// SIMATIC STEP 7 (V5.x) project waterplant
// CPU: CPU 314C-2 DP
// station: Hardware
// station: SIMATIC 300(1)
// station: P_ADR_BUS
// station: P_ADR_BUS
// station: Configuration
// program: S7 Program(1)

SYMBOL_TABLE
"S5TI_TIM"	FC 33	FC 33	// S5 Time to IEC Time
"TIM_S5TI"	FC 40	FC 40	// IEC Time to S5 Time
"SCALE"	FC 105	FC 105	// Scaling Values
"start system"	I 0.0	BOOL
"LEVsensor Raw tank"	I 0.1	BOOL
"raw pump run feedback"	I 0.2	BOOL
"low filter tank1"	I 0.3	BOOL
"high filter tank1"	I 0.4	BOOL
"low filter tank2"	I 0.5	BOOL
"emergency pressed"	I 0.6	BOOL
"sludge H-sensor tank"	I 0.7	BOOL
"LEVsensor flash mixer"	I 1.0	BOOL
"LEVsensor slow mixer"	I 1.1	BOOL
"LEVsenclarifier buttom"	I 1.2	BOOL
"sludge L-sensor tank"	I 1.3	BOOL
"led photo sensor"	I 1.4	BOOL
"service intake"	I 1.5	BOOL
"flash mixer feedback"	I 2.0	BOOL
"slow mixer feedback"	I 2.1	BOOL
"clarifier feedback"	I 2.2	BOOL
"blower feedback"	I 2.3	BOOL
"wash water feedback"	I 2.4	BOOL
"flash mixer over sensor"	I 2.5	BOOL
"PLC OK"	M 0.0	BOOL
"reset sludge clarifier"	M 0.1	BOOL
"sludge clarifier relay"	M 0.2	BOOL
"test clarifier from scad"	M 0.3	BOOL
"test raw pump scada"	M 0.4	BOOL
"test flash mixer scada"	M 0.5	BOOL
"test slow mixer scada"	M 0.6	BOOL
"test sludge pump scada"	M 0.7	BOOL
"sludge pipe color scada"	M 1.0	BOOL
"led test from scada"	M 1.1	BOOL
"air valve relay"	M 1.2	BOOL
"air valve test scada"	M 1.3	BOOL
"traet pipe color"	M 1.4	BOOL
"wash water relay"	M 1.5	BOOL
"wash water test scada"	M 1.6	BOOL
"zero washing time messag"	M 1.7	BOOL
"sludge time message"	M 2.0	BOOL
"reset alarm scada"	M 2.1	BOOL
"reset hardware alarm"	M 2.2	BOOL
"alarm on scada"	M 2.3	BOOL
"factory reset scada"	M 2.4	BOOL
"system run for scada"	M 2.5	BOOL
"filter tank H-L relay"	M 2.6	BOOL
"sludge pump relay"	M 2.7	BOOL
"raw pump feedback alarm"	M 3.0	BOOL
"force stop raw pump"	M 3.1	BOOL
"force stop AL2SO4"	M 3.2	BOOL
"force stop flash mixer"	M 3.3	BOOL
"force stop slow mixer"	M 3.4	BOOL
"force stop sludge pump"	M 3.5	BOOL
"force stop clarifier"	M 3.6	BOOL
"air blower force stop"	M 3.7	BOOL
"wash pump force stop"	M 4.0	BOOL
"alarm on scada relay"	M 4.1	BOOL
"air valve relay 2"	M 4.2	BOOL
"wash water relay 2"	M 4.3	BOOL
"force stop light"	M 4.4	BOOL
"flash mixer over"	M 4.6	BOOL
"zero analog bibolar"	M 5.0	BOOL
"flash mixer tank full"	M 5.1	BOOL
"slow mixer full tank"	M 5.2	BOOL
"flash feedback  alarm"	M 5.3	BOOL
"start reverse now scada"	M 5.5	BOOL
"restart reverse wash sca"	M 5.6	BOOL
"No restert scada"	M 5.7	BOOL
"No restart marker"	M 6.0	BOOL
"reverse wash wait messag"	M 6.1	BOOL
"sludge tank filling"	M 6.2	BOOL
"emeergency mode for scad"	M 6.3	BOOL
"start now marker"	M 6.4	BOOL
"reverse wash has started"	M 6.6	BOOL
"slow feedback alarm"	M 6.7	BOOL
"clarifier feedback alarm"	M 7.0	BOOL
"blower feedback alarm"	M 7.1	BOOL
"wash feedback alarm"	M 7.2	BOOL
"flash over flow alarm"	M 7.3	BOOL
"y.restart rev wash scada"	M 8.0	BOOL
"reverser timer reminder"	MD 210	DWORD
"rev wash reminder scada"	MD 212	DWORD
"sludge clarifier off sca"	MW 50	WORD
"sludge clarifier on sca"	MW 80	WORD
"reverse wash time scada"	MW 150	WORD
"voltage sensor analoge"	PIW 3	WORD
"current sensor analoge"	PIW 5	WORD
"raw pump"	Q 0.0	BOOL
"AL2SO4 valve"	Q 0.1	BOOL
"flash mixer"	Q 0.2	BOOL
"slow mixer"	Q 0.3	BOOL
"sludge motor clarifier"	Q 0.4	BOOL
"enter valve filter1"	Q 0.5	BOOL
"enter valve filter2"	Q 0.6	BOOL
"treat1"	Q 0.7	BOOL
"treat2"	Q 1.0	BOOL
"air valve1"	Q 1.1	BOOL
"wash water1"	Q 1.2	BOOL
"sludge pump"	Q 1.3	BOOL
"alarm"	Q 1.4	BOOL
"led"	Q 1.5	BOOL
"sludge valve filter1"	Q 1.6	BOOL
"sludge valve filter2"	Q 1.7	BOOL
"TON"	SFB 4	SFB 4	// Generate an On Delay
"AL2SO4 open time"	T 1	TIMER
"clarifier off time"	T 2	TIMER
"clarifier on time"	T 3	TIMER
"high treat tank dist"	T 4	TIMER
"wash timer process"	T 5	TIMER
"air valve timer"	T 6	TIMER
"before wash time"	T 8	TIMER	// delay time before start washing
"treat1 dist"	T 9	TIMER
"enter valve 1 delay time"	T 10	TIMER
"slow feedback timer"	T 11	TIMER
"delay time before alarm"	T 12	TIMER
"factory reset timer"	T 13	TIMER
"start system timer"	T 14	TIMER
"clarifier feedback timer"	T 15	TIMER
"blower feedback timer"	T 16	TIMER
"sludge pump force stop t"	T 17	TIMER
"clarifier force stop t"	T 18	TIMER
"raw pump force stop t"	T 19	TIMER
"clarifier before start t"	T 20	TIMER
"timer before wash proces"	T 21	TIMER
"wash feedback timer"	T 22	TIMER
"treat 2 dist."	T 23	TIMER
"flash mixer feedback tim"	T 24	TIMER
"raw pump feedback timer"	T 25	TIMER
"enter valve 2 timer"	T 26	TIMER
"before restart message"	T 30	TIMER
"rewash wait alarm timer"	T 31	TIMER
END_SYMBOL_TABLE

// FC 33: know-how protected block, not included

// FC 40: know-how protected block, not included

// FC 105: know-how protected block, not included

ORGANIZATION_BLOCK OB 1
TITLE = "Main Program Sweep (Cycle)"
VERSION : 0.1
VAR_TEMP
  OB1_EV_CLASS : BYTE ;	//Bits 0-3 = 1 (Coming event), Bits 4-7 = 1 (Event class 1)
  OB1_SCAN_1 : BYTE ;	//1 (Cold restart scan 1 of OB 1), 3 (Scan 2-n of OB 1)
  OB1_PRIORITY : BYTE ;	//Priority of OB Execution
  OB1_OB_NUMBR : BYTE ;	//1 (Organization block 1, OB1)
  OB1_RESERVED_1 : BYTE ;	//Reserved for system
  OB1_RESERVED_2 : BYTE ;	//Reserved for system
  OB1_PREV_CYCLE : INT ;	//Cycle time of previous OB1 scan (milliseconds)
  OB1_MIN_CYCLE : INT ;	//Minimum cycle time of OB1 (milliseconds)
  OB1_MAX_CYCLE : INT ;	//Maximum cycle time of OB1 (milliseconds)
  OB1_DATE_TIME : DATE_AND_TIME ;	//Date and time OB1 started
END_VAR
BEGIN
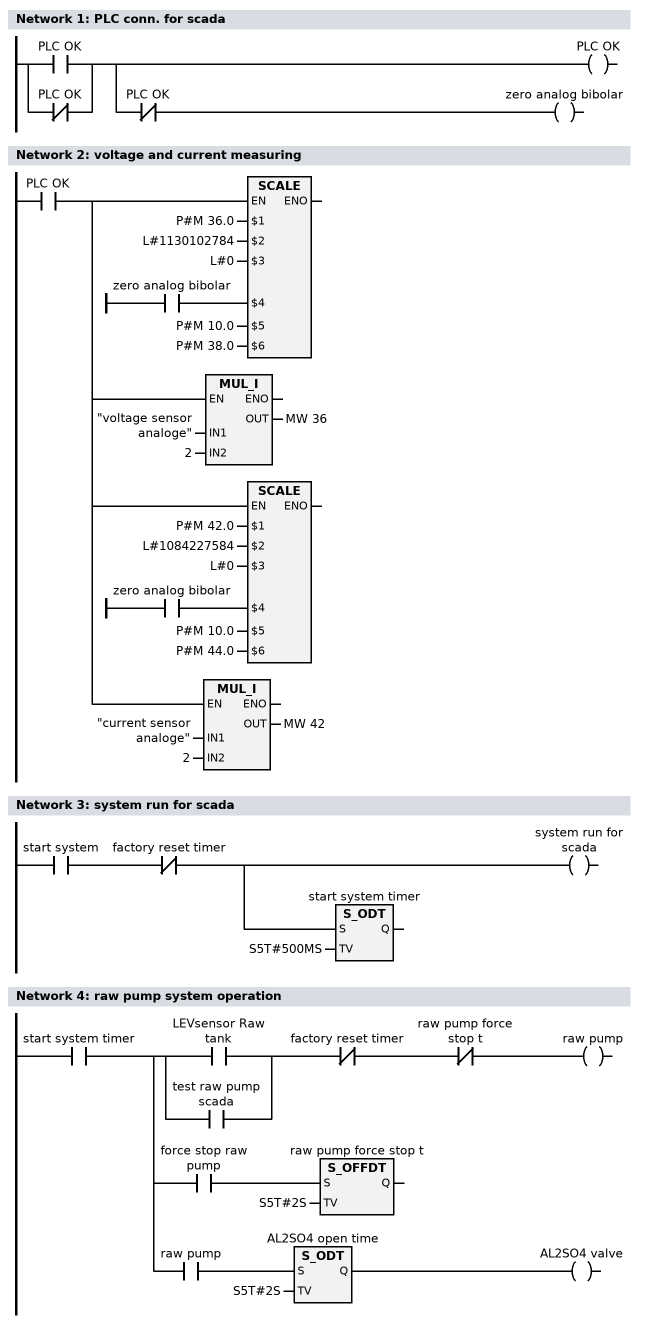
NETWORK
TITLE = PLC conn. for scada
      O     "PLC OK";
      ON    "PLC OK";
      =     L 240.0;
      A     L 240.0;
      BLD   102;
      =     "PLC OK";
      A     L 240.0;
      AN    "PLC OK";
      =     "zero analog bibolar";
NETWORK
TITLE = voltage and current measuring
      A     "PLC OK";
      =     L 240.0;
      A     "zero analog bibolar";
      =     L 240.1;
      BLD   103;
      A     L 240.0;
      JNB   _001;
      CALL  "SCALE" (
           $1                       := P#M 36.0,
           $2                       := L#1130102784,
           $3                       := L#0,
           $4                       := L 240.1,
           $5                       := P#M 10.0,
           $6                       := P#M 38.0);
_001: NOP   0;
      A     L 240.0;
      JNB   _002;
      L     "voltage sensor analoge";
      L     2;
      *I;
      T     MW 36;
_002: NOP   0;
      A     "zero analog bibolar";
      =     L 240.1;
      BLD   103;
      A     L 240.0;
      JNB   _003;
      CALL  "SCALE" (
           $1                       := P#M 42.0,
           $2                       := L#1084227584,
           $3                       := L#0,
           $4                       := L 240.1,
           $5                       := P#M 10.0,
           $6                       := P#M 44.0);
_003: NOP   0;
      A     L 240.0;
      JNB   _004;
      L     "current sensor analoge";
      L     2;
      *I;
      T     MW 42;
_004: NOP   0;
NETWORK
TITLE = system run for scada
      A     "start system";
      AN    "factory reset timer";
      =     L 240.0;
      A     L 240.0;
      BLD   102;
      =     "system run for scada";
      A     L 240.0;
      L     S5T#500MS;
      SD    "start system timer";
      NOP   0;
      NOP   0;
      NOP   0;
      NOP   0;
NETWORK
TITLE = raw pump system operation
      A     "start system timer";
      =     L 240.0;
      A     L 240.0;
      A(;
      O     "LEVsensor Raw tank";
      O     "test raw pump scada";
      );
      AN    "factory reset timer";
      AN    "raw pump force stop t";
      =     "raw pump";
      A     L 240.0;
      A     "force stop raw pump";
      L     S5T#2S;
      SF    "raw pump force stop t";
      NOP   0;
      NOP   0;
      NOP   0;
      NOP   0;
      A     L 240.0;
      A     "raw pump";
      L     S5T#2S;
      SD    "AL2SO4 open time";
      NOP   0;
      NOP   0;
      NOP   0;
      A     "AL2SO4 open time";
      =     "AL2SO4 valve";
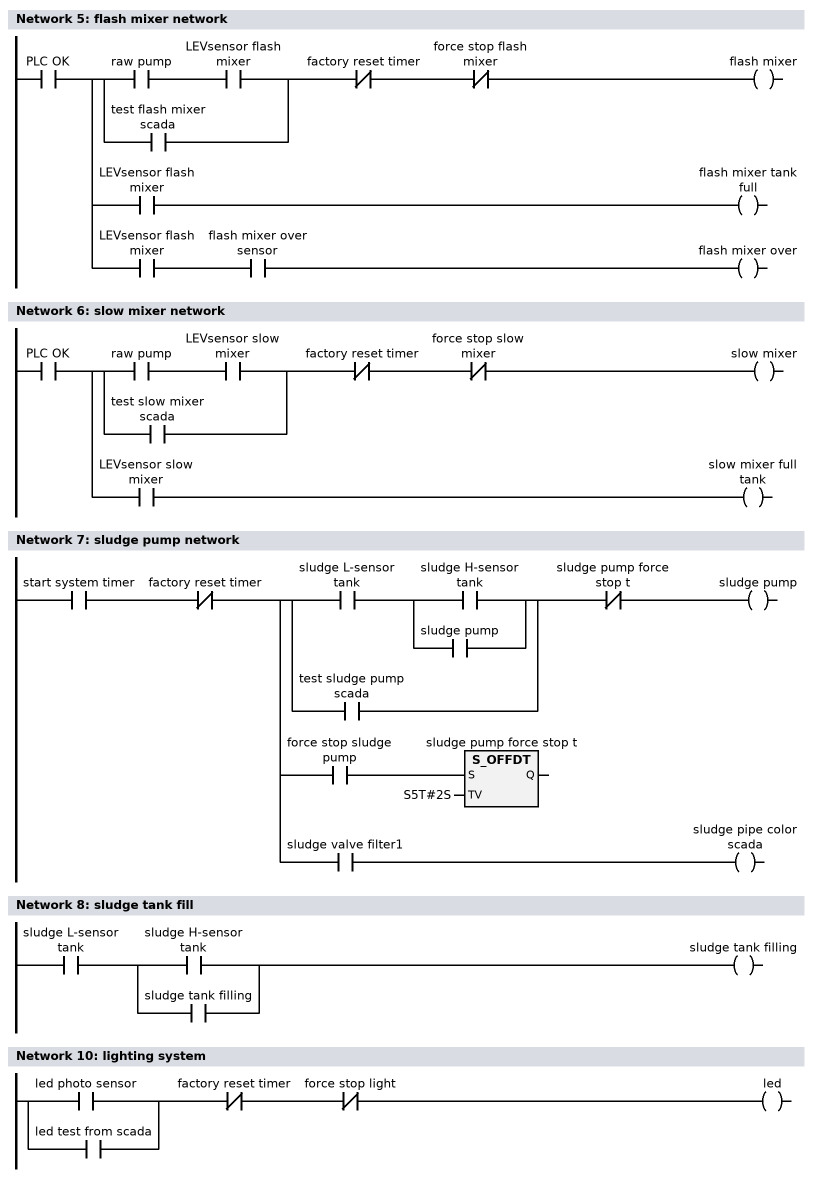
NETWORK
TITLE = flash mixer network
      A     "PLC OK";
      =     L 240.0;
      A     L 240.0;
      A(;
      A     "raw pump";
      A     "LEVsensor flash mixer";
      O     "test flash mixer scada";
      );
      AN    "factory reset timer";
      AN    "force stop flash mixer";
      =     "flash mixer";
      A     L 240.0;
      A     "LEVsensor flash mixer";
      =     "flash mixer tank full";
      A     L 240.0;
      A     "LEVsensor flash mixer";
      A     "flash mixer over sensor";
      =     "flash mixer over";
NETWORK
TITLE = slow mixer network
      A     "PLC OK";
      =     L 240.0;
      A     L 240.0;
      A(;
      A     "raw pump";
      A     "LEVsensor slow mixer";
      O     "test slow mixer scada";
      );
      AN    "factory reset timer";
      AN    "force stop slow mixer";
      =     "slow mixer";
      A     L 240.0;
      A     "LEVsensor slow mixer";
      =     "slow mixer full tank";
NETWORK
TITLE = sludge pump network
      A     "start system timer";
      AN    "factory reset timer";
      =     L 240.0;
      A     L 240.0;
      A(;
      A     "sludge L-sensor tank";
      A(;
      O     "sludge H-sensor tank";
      O     "sludge pump";
      );
      O     "test sludge pump scada";
      );
      AN    "sludge pump force stop t";
      =     "sludge pump";
      A     L 240.0;
      A     "force stop sludge pump";
      L     S5T#2S;
      SF    "sludge pump force stop t";
      NOP   0;
      NOP   0;
      NOP   0;
      NOP   0;
      A     L 240.0;
      A     "sludge valve filter1";
      =     "sludge pipe color scada";
NETWORK
TITLE = sludge tank fill
      A     "sludge L-sensor tank";
      A(;
      O     "sludge H-sensor tank";
      O     "sludge tank filling";
      );
      =     "sludge tank filling";
NETWORK
TITLE = sludge motor clarifier timer operation
      A     "start system timer";
      =     L 240.0;
      A     L 240.0;
      A     "raw pump";
      A     "LEVsenclarifier buttom";
      AN    "factory reset timer";
      =     L 240.1;
      A(;
      A     L 240.1;
      A(;
      L     "sludge clarifier off sca";
      L     0;
      >I;
      );
      A(;
      L     "sludge clarifier on sca";
      L     0;
      >I;
      );
      L     S5T#50MS;
      SD    "clarifier before start t";
      NOP   0;
      NOP   0;
      NOP   0;
      A     "clarifier before start t";
      );
      AN    "clarifier on time";
      L     MW 54;
      SD    "clarifier off time";
      NOP   0;
      NOP   0;
      LC    "clarifier off time";
      T     MW 58;
      NOP   0;
      A(;
      A(;
      A     L 240.1;
      JNB   _005;
      CALL  "S5TI_TIM" (
           $1                       := P#M 58.0,
           $2                       := P#M 62.0);
_005: A     BR;
      );
      JNB   _006;
      L     MD 62;
      DTR;
      T     MD 66;
      SET;
      SAVE;
      CLR;
_006: A     BR;
      );
      JNB   _007;
      L     MD 66;
      L     1.000000e+03;
      /R;
      T     MD 70;
_007: NOP   0;
      A     L 240.1;
      A     "clarifier off time";
      L     MW 84;
      SD    "clarifier on time";
      NOP   0;
      NOP   0;
      LC    "clarifier on time";
      T     MW 88;
      NOP   0;
      A(;
      A(;
      A     L 240.1;
      JNB   _008;
      CALL  "S5TI_TIM" (
           $1                       := P#M 88.0,
           $2                       := P#M 92.0);
_008: A     BR;
      );
      JNB   _009;
      L     MD 92;
      DTR;
      T     MD 96;
      SET;
      SAVE;
      CLR;
_009: A     BR;
      );
      JNB   _00a;
      L     MD 96;
      L     1.000000e+03;
      /R;
      T     MD 100;
_00a: NOP   0;
      A     L 240.1;
      A(;
      L     "sludge clarifier off sca";
      L     0;
      <>I;
      );
      A(;
      L     "sludge clarifier on sca";
      L     0;
      <>I;
      );
      A     "clarifier off time";
      AN    "clarifier on time";
      =     "sludge clarifier relay";
      A(;
      A(;
      A     L 240.0;
      JNB   _00b;
      L     "sludge clarifier off sca";
      ITD;
      T     LD 50;
      SET;
      SAVE;
      CLR;
_00b: A     BR;
      );
      JNB   _00c;
      L     LD 50;
      L     1000;
      *D;
      T     LD 54;
      AN    OV;
      SAVE;
      CLR;
_00c: A     BR;
      );
      JNB   _00d;
      CALL  "TIM_S5TI" (
           $1                       := P#L 54.0,
           $2                       := P#M 54.0);
_00d: NOP   0;
      A(;
      A(;
      A     L 240.0;
      JNB   _00e;
      L     "sludge clarifier on sca";
      ITD;
      T     LD 80;
      SET;
      SAVE;
      CLR;
_00e: A     BR;
      );
      JNB   _00f;
      L     LD 80;
      L     1000;
      *D;
      T     LD 84;
      AN    OV;
      SAVE;
      CLR;
_00f: A     BR;
      );
      JNB   _010;
      CALL  "TIM_S5TI" (
           $1                       := P#L 84.0,
           $2                       := P#M 84.0);
_010: NOP   0;
      A     L 240.0;
      A     "force stop clarifier";
      L     S5T#2S;
      SF    "clarifier force stop t";
      NOP   0;
      NOP   0;
      NOP   0;
      NOP   0;
      A     L 240.0;
      A(;
      O     "sludge clarifier relay";
      O     "test clarifier from scad";
      );
      AN    "clarifier force stop t";
      =     "sludge motor clarifier";
      A     L 240.0;
      A     "reset sludge clarifier";
      =     L 240.1;
      A     L 240.1;
      JNB   _011;
      L     0;
      T     "sludge clarifier off sca";
_011: NOP   0;
      A     L 240.1;
      JNB   _012;
      L     0;
      T     "sludge clarifier on sca";
_012: NOP   0;
NETWORK
TITLE = lighting system
      A(;
      O     "led photo sensor";
      O     "led test from scada";
      );
      AN    "factory reset timer";
      AN    "force stop light";
      =     "led";
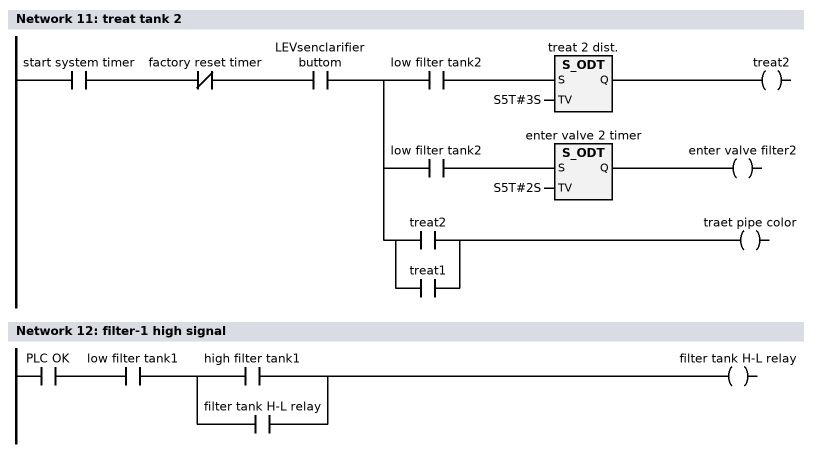
NETWORK
TITLE = treat tank 2
      A     "start system timer";
      AN    "factory reset timer";
      A     "LEVsenclarifier buttom";
      =     L 240.0;
      A     L 240.0;
      A     "low filter tank2";
      L     S5T#3S;
      SD    "treat 2 dist.";
      NOP   0;
      NOP   0;
      NOP   0;
      A     "treat 2 dist.";
      =     "treat2";
      A     L 240.0;
      A     "low filter tank2";
      L     S5T#2S;
      SD    "enter valve 2 timer";
      NOP   0;
      NOP   0;
      NOP   0;
      A     "enter valve 2 timer";
      =     "enter valve filter2";
      A     L 240.0;
      A(;
      O     "treat2";
      O     "treat1";
      );
      =     "traet pipe color";
NETWORK
TITLE = filter-1 high signal
      A     "PLC OK";
      A     "low filter tank1";
      A(;
      O     "high filter tank1";
      O     "filter tank H-L relay";
      );
      =     "filter tank H-L relay";
NETWORK
TITLE = treat tank 1
      A     "start system timer";
      =     L 240.0;
      A     L 240.0;
      AN    "factory reset timer";
      A     "LEVsenclarifier buttom";
      =     L 240.1;
      A     L 240.1;
      AN    "high treat tank dist";
      L     S5T#2S;
      SD    "enter valve 1 delay time";
      NOP   0;
      NOP   0;
      NOP   0;
      A     "enter valve 1 delay time";
      =     "enter valve filter1";
      A     L 240.1;
      A     "filter tank H-L relay";
      L     S5T#2S;
      SD    "high treat tank dist";
      NOP   0;
      NOP   0;
      NOP   0;
      NOP   0;
      A     L 240.1;
      A(;
      O     "enter valve filter1";
      O     "No restart marker";
      );
      A     "low filter tank1";
      A(;
      ON    "high treat tank dist";
      O     "No restart marker";
      );
      AN    "factory reset timer";
      L     S5T#2S;
      SD    "treat1 dist";
      NOP   0;
      NOP   0;
      NOP   0;
      A     "treat1 dist";
      =     "treat1";
      A     L 240.1;
      A     "wash timer process";
      =     L 240.2;
      A     L 240.2;
      L     S5T#500MS;
      SD    "before restart message";
      NOP   0;
      NOP   0;
      NOP   0;
      NOP   0;
      A     L 240.2;
      AN    "No restart marker";
      L     S5T#10S;
      SD    "rewash wait alarm timer";
      NOP   0;
      NOP   0;
      NOP   0;
      NOP   0;
      A     L 240.1;
      A(;
      A     "before restart message";
      A     "No restert scada";
      O     "No restart marker";
      O     "rewash wait alarm timer";
      );
      A     "low filter tank1";
      =     "No restart marker";
      A     L 240.1;
      A     "before restart message";
      AN    "No restart marker";
      =     "restart reverse wash sca";
      A     L 240.1;
      A(;
      O     "start reverse now scada";
      O     "start now marker";
      );
      AN    "wash timer process";
      =     "start now marker";
      A     L 240.1;
      A(;
      O     "high treat tank dist";
      O     "start now marker";
      );
      A(;
      L     "reverse wash time scada";
      L     0;
      >I;
      );
      L     S5T#1S;
      SD    "timer before wash proces";
      NOP   0;
      NOP   0;
      NOP   0;
      A     "timer before wash proces";
      =     L 240.2;
      A     L 240.2;
      AN    "y.restart rev wash scada";
      L     S5T#1S;
      SD    "before wash time";
      NOP   0;
      NOP   0;
      NOP   0;
      A     "before wash time";
      =     L 240.3;
      A     L 240.3;
      A     "sludge valve filter1";
      L     MW 154;
      SD    "wash timer process";
      NOP   0;
      NOP   0;
      LC    "wash timer process";
      T     MW 200;
      NOP   0;
      A     L 240.3;
      JNB   _013;
      L     MW 200;
      BTI;
      T     LW 226;
      SET;
      SAVE;
      CLR;
_013: A     BR;
      =     L 240.4;
      A     L 240.4;
      A(;
      L     "reverse wash time scada";
      L     99;
      <=I;
      );
      A     "PLC OK";
      =     L 240.5;
      A     L 240.5;
      A(;
      L     LW 226;
      L     LW 220;
      >I;
      );
      =     "air valve relay";
      A     L 240.5;
      AN    "wash timer process";
      A(;
      L     LW 226;
      L     LW 224;
      <=I;
      );
      =     "wash water relay";
      A     L 240.4;
      A(;
      L     "reverse wash time scada";
      L     99;
      >I;
      );
      A     "PLC OK";
      =     L 240.5;
      A     L 240.5;
      A(;
      L     LW 226;
      L     LW 236;
      >I;
      );
      =     "air valve relay 2";
      A     L 240.5;
      AN    "wash timer process";
      A(;
      L     LW 226;
      L     LW 238;
      <=I;
      );
      =     "wash water relay 2";
      A     L 240.2;
      BLD   102;
      =     "sludge valve filter1";
      A(;
      A(;
      A     L 240.0;
      JNB   _014;
      L     "reverse wash time scada";
      ITD;
      T     LD 150;
      SET;
      SAVE;
      CLR;
_014: A     BR;
      );
      JNB   _015;
      L     LD 150;
      L     1000;
      *D;
      T     LD 154;
      AN    OV;
      SAVE;
      CLR;
_015: A     BR;
      );
      JNB   _016;
      CALL  "TIM_S5TI" (
           $1                       := P#L 154.0,
           $2                       := P#M 154.0);
_016: NOP   0;
      A(;
      A(;
      A     L 240.0;
      JNB   _017;
      CALL  "S5TI_TIM" (
           $1                       := P#M 200.0,
           $2                       := P#M 204.0);
_017: A     BR;
      );
      JNB   _018;
      L     MD 204;
      DTR;
      T     MD 208;
      SET;
      SAVE;
      CLR;
_018: A     BR;
      );
      JNB   _019;
      L     MD 208;
      L     1.000000e+03;
      /R;
      T     "rev wash reminder scada";
_019: NOP   0;
      A     L 240.0;
      A(;
      L     "reverse wash time scada";
      L     99;
      <=I;
      );
      JNB   _01a;
      L     "reverse wash time scada";
      L     10;
      *I;
      T     LW 216;
      AN    OV;
      SAVE;
      CLR;
_01a: A     BR;
      =     L 240.1;
      A(;
      A     L 240.1;
      JNB   _01b;
      L     LW 216;
      L     3;
      /I;
      T     LW 218;
      AN    OV;
      SAVE;
      CLR;
_01b: A     BR;
      );
      JNB   _01c;
      L     LW 216;
      L     LW 218;
      -I;
      T     LW 220;
_01c: NOP   0;
      A(;
      A     L 240.1;
      JNB   _01d;
      L     LW 216;
      L     6;
      /I;
      T     LW 222;
      AN    OV;
      SAVE;
      CLR;
_01d: A     BR;
      );
      JNB   _01e;
      L     LW 216;
      L     LW 222;
      -I;
      T     LW 224;
_01e: NOP   0;
      A     L 240.0;
      A(;
      L     "reverse wash time scada";
      L     99;
      >I;
      );
      JNB   _01f;
      L     "reverse wash time scada";
      L     1;
      *I;
      T     LW 230;
      AN    OV;
      SAVE;
      CLR;
_01f: A     BR;
      =     L 240.1;
      A(;
      A     L 240.1;
      JNB   _020;
      L     LW 230;
      L     3;
      /I;
      T     LW 232;
      AN    OV;
      SAVE;
      CLR;
_020: A     BR;
      );
      JNB   _021;
      L     LW 230;
      L     LW 232;
      -I;
      T     LW 236;
_021: NOP   0;
      A(;
      A     L 240.1;
      JNB   _022;
      L     LW 230;
      L     6;
      /I;
      T     LW 234;
      AN    OV;
      SAVE;
      CLR;
_022: A     BR;
      );
      JNB   _023;
      L     LW 230;
      L     LW 234;
      -I;
      T     LW 238;
_023: NOP   0;
      A     L 240.0;
      A(;
      O     "air valve relay";
      O     "air valve relay 2";
      O     "air valve test scada";
      );
      AN    "factory reset timer";
      AN    "air blower force stop";
      =     "air valve1";
      A     L 240.0;
      A(;
      O     "wash water relay";
      O     "wash water relay 2";
      O     "wash water test scada";
      );
      AN    "factory reset timer";
      AN    "wash pump force stop";
      =     "wash water1";
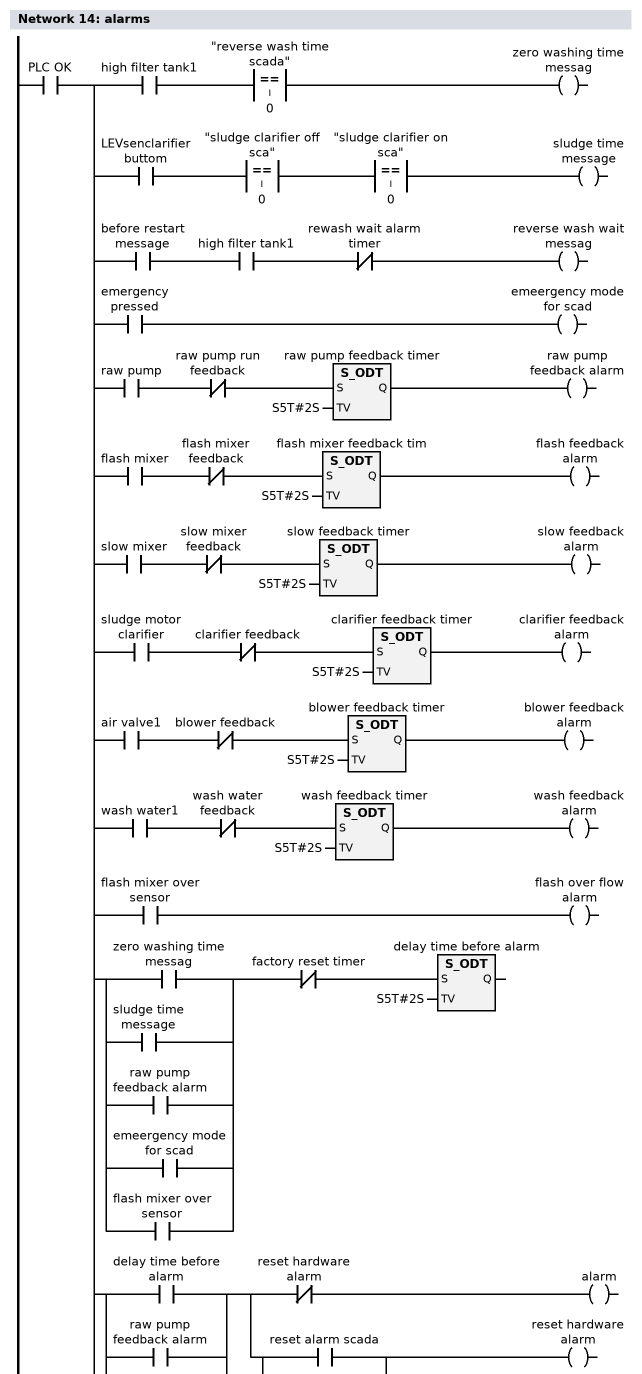
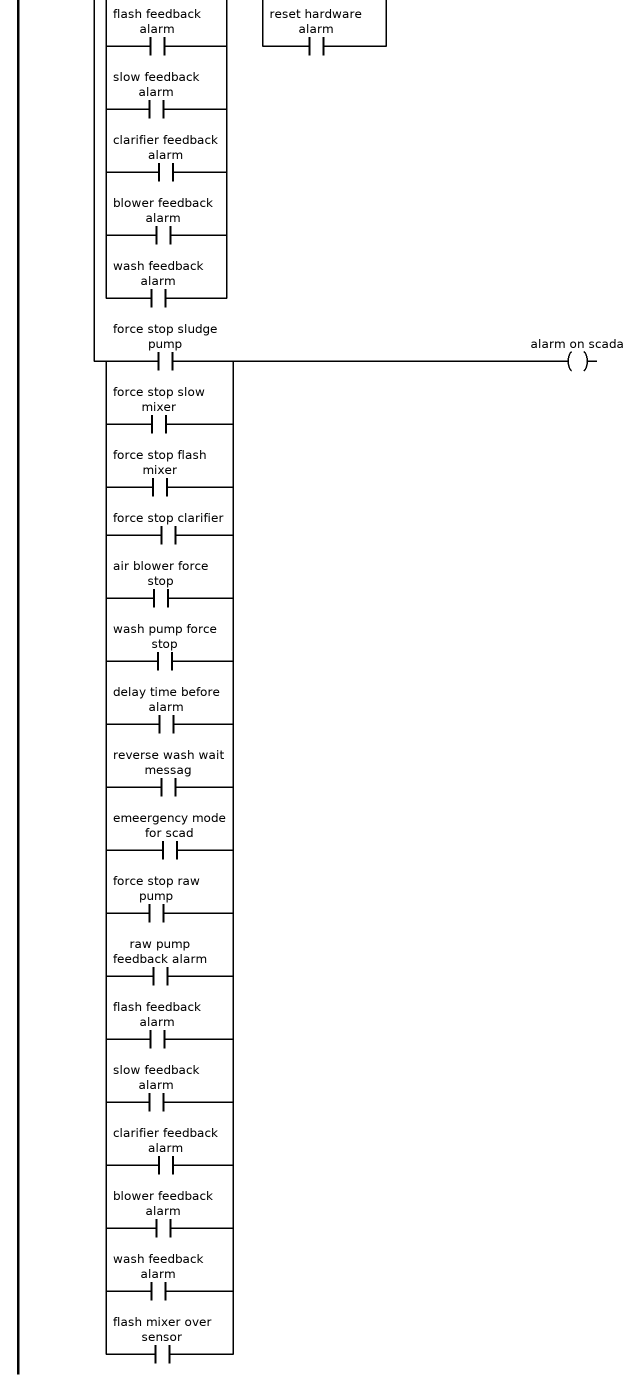
NETWORK
TITLE = alarms
      A     "PLC OK";
      =     L 240.0;
      A     L 240.0;
      A     "high filter tank1";
      A(;
      L     "reverse wash time scada";
      L     0;
      ==I;
      );
      =     "zero washing time messag";
      A     L 240.0;
      A     "LEVsenclarifier buttom";
      A(;
      L     "sludge clarifier off sca";
      L     0;
      ==I;
      );
      A(;
      L     "sludge clarifier on sca";
      L     0;
      ==I;
      );
      =     "sludge time message";
      A     L 240.0;
      A     "before restart message";
      A     "high filter tank1";
      AN    "rewash wait alarm timer";
      =     "reverse wash wait messag";
      A     L 240.0;
      A     "emergency pressed";
      =     "emeergency mode for scad";
      A     L 240.0;
      A     "raw pump";
      AN    "raw pump run feedback";
      L     S5T#2S;
      SD    "raw pump feedback timer";
      NOP   0;
      NOP   0;
      NOP   0;
      A     "raw pump feedback timer";
      =     "raw pump feedback alarm";
      A     L 240.0;
      A     "flash mixer";
      AN    "flash mixer feedback";
      L     S5T#2S;
      SD    "flash mixer feedback tim";
      NOP   0;
      NOP   0;
      NOP   0;
      A     "flash mixer feedback tim";
      =     "flash feedback  alarm";
      A     L 240.0;
      A     "slow mixer";
      AN    "slow mixer feedback";
      L     S5T#2S;
      SD    "slow feedback timer";
      NOP   0;
      NOP   0;
      NOP   0;
      A     "slow feedback timer";
      =     "slow feedback alarm";
      A     L 240.0;
      A     "sludge motor clarifier";
      AN    "clarifier feedback";
      L     S5T#2S;
      SD    "clarifier feedback timer";
      NOP   0;
      NOP   0;
      NOP   0;
      A     "clarifier feedback timer";
      =     "clarifier feedback alarm";
      A     L 240.0;
      A     "air valve1";
      AN    "blower feedback";
      L     S5T#2S;
      SD    "blower feedback timer";
      NOP   0;
      NOP   0;
      NOP   0;
      A     "blower feedback timer";
      =     "blower feedback alarm";
      A     L 240.0;
      A     "wash water1";
      AN    "wash water feedback";
      L     S5T#2S;
      SD    "wash feedback timer";
      NOP   0;
      NOP   0;
      NOP   0;
      A     "wash feedback timer";
      =     "wash feedback alarm";
      A     L 240.0;
      A     "flash mixer over sensor";
      =     "flash over flow alarm";
      A     L 240.0;
      A(;
      O     "zero washing time messag";
      O     "sludge time message";
      O     "raw pump feedback alarm";
      O     "emeergency mode for scad";
      O     "flash mixer over sensor";
      );
      AN    "factory reset timer";
      L     S5T#2S;
      SD    "delay time before alarm";
      NOP   0;
      NOP   0;
      NOP   0;
      NOP   0;
      A     L 240.0;
      A(;
      O     "delay time before alarm";
      O     "raw pump feedback alarm";
      O     "flash feedback  alarm";
      O     "slow feedback alarm";
      O     "clarifier feedback alarm";
      O     "blower feedback alarm";
      O     "wash feedback alarm";
      );
      =     L 240.1;
      A     L 240.1;
      AN    "reset hardware alarm";
      =     "alarm";
      A     L 240.1;
      A(;
      O     "reset alarm scada";
      O     "reset hardware alarm";
      );
      =     "reset hardware alarm";
      A     L 240.0;
      A(;
      O     "force stop sludge pump";
      O     "force stop slow mixer";
      O     "force stop flash mixer";
      O     "force stop clarifier";
      O     "air blower force stop";
      O     "wash pump force stop";
      O     "delay time before alarm";
      O     "reverse wash wait messag";
      O     "emeergency mode for scad";
      O     "force stop raw pump";
      O     "raw pump feedback alarm";
      O     "flash feedback  alarm";
      O     "slow feedback alarm";
      O     "clarifier feedback alarm";
      O     "blower feedback alarm";
      O     "wash feedback alarm";
      O     "flash mixer over sensor";
      );
      =     "alarm on scada";
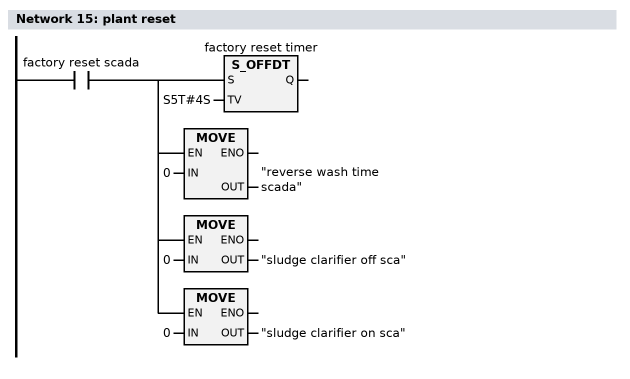
NETWORK
TITLE = plant reset 
      A     "factory reset scada";
      =     L 240.0;
      A     L 240.0;
      L     S5T#4S;
      SF    "factory reset timer";
      NOP   0;
      NOP   0;
      NOP   0;
      NOP   0;
      A     L 240.0;
      JNB   _024;
      L     0;
      T     "reverse wash time scada";
_024: NOP   0;
      A     L 240.0;
      JNB   _025;
      L     0;
      T     "sludge clarifier off sca";
_025: NOP   0;
      A     L 240.0;
      JNB   _026;
      L     0;
      T     "sludge clarifier on sca";
_026: NOP   0;
END_ORGANIZATION_BLOCK
